PROGRAM Vac_Ctrl
VAR
    Vacuums     : ARRAY[1..4] OF ST_Vacuum;
    VacuumFB    : ARRAY[1..4] OF FB_VacuumControl;
    bResetAll   : BOOL;
    i           : INT;
END_VAR








(* 输出 *)
//Y000212 := stVac[1].qVacuumValve;
//Y000213 := stVac[1].qReleaseValve;
//Y000214 := stVac[2].qVacuumValve;
//Y000215 := stVac[2].qReleaseValve;

END_PROGRAM

(* stored: Version 1.1.0.1, ProductVersion 3.1.4024.12
   POU Vac_Ctrl: Id {b4ee8d84-c47f-41eb-8d8b-f0b2e844f0f1}, SpecialFunc None *)
